FUNCTION_BLOCK CompositeBlockWithoutConnections
  FBS
    BaseBlock1 : BaseBlock;
    EA_RightPublishSubscribeAdapter : EA_RightPublishSubscribeAdapter;
    Publish_Right_EA : PUBLISH_5;
    Subscribe_Right_EA : SUBSCRIBE_5;
    EA_network2 : EA_network2;
  END_FBS
  EVENT_CONNECTIONS
    EA_RightPublishSubscribeAdapter.REQ TO Publish_Right_EA.REQ;
    Subscribe_Right_EA.IND TO EA_RightPublishSubscribeAdapter.IND;
  END_CONNECTIONS
  DATA_CONNECTIONS
    EA_RightPublishSubscribeAdapter.I_E_number TO Publish_Right_EA.SD_1;
    EA_RightPublishSubscribeAdapter.I_data1 TO Publish_Right_EA.SD_2;
    EA_RightPublishSubscribeAdapter.I_data2 TO Publish_Right_EA.SD_3;
    EA_RightPublishSubscribeAdapter.N_O_data1 TO Publish_Right_EA.SD_4;
    EA_RightPublishSubscribeAdapter.N_O_data2 TO Publish_Right_EA.SD_5;
    Subscribe_Right_EA.RD_1 TO EA_RightPublishSubscribeAdapter.O_E_number;
    Subscribe_Right_EA.RD_2 TO EA_RightPublishSubscribeAdapter.O_data1;
    Subscribe_Right_EA.RD_3 TO EA_RightPublishSubscribeAdapter.O_data2;
    Subscribe_Right_EA.RD_4 TO EA_RightPublishSubscribeAdapter.N_I_data1;
    Subscribe_Right_EA.RD_5 TO EA_RightPublishSubscribeAdapter.N_I_data2;
  END_CONNECTIONS
  ADAPTER_CONNECTIONS
    EA_RightPublishSubscribeAdapter.plug TO EA_network2.socket;
    EA_network2.plug TO BaseBlock1.socket;
  END_CONNECTIONS
END_FUNCTION_BLOCK
